TYPE ST_ModuleFileConfig :
STRUCT
	Enabled : BOOL;
	Slot : UINT;
	Id : UDINT;
	ModuleType : STRING(16);
	InputMappingCount : UINT;
	InputMappings : ARRAY[1..Param_Config.MaxModuleMappings] OF ST_MappingFileConfig;
	OutputMappingCount : UINT;
	OutputMappings : ARRAY[1..Param_Config.MaxModuleMappings] OF ST_MappingFileConfig;
	ReferenceBindingCount : UINT;
	ReferenceBindings : ARRAY[1..Param_Config.MaxModuleReferenceBindings] OF ST_ReferenceBindingFileConfig;
	VariableCount : UINT;
	VariableList : ARRAY[1..Param_Config.MaxModuleVariable] OF ST_ConfigVariableInfo;
	AlarmCount : UINT;
	AlarmList : ARRAY[1..Param_Config.MaxConfiguredAlarmsPerModule] OF ST_ConfigAlarmInfo;
END_STRUCT
END_TYPE

(* stored: Version 1.1.0.1, ProductVersion 3.1.4026.18
   DUT ST_ModuleFileConfig: Id {c62416ff-7f4d-4f67-a53f-e338d36967f9} *)
